_CFC_ (* Continuous Function Chart, elements in execution order *)
(* GYM *)
(* CINEMA *)
(* SHOWER *)
(* SPHERE *)
(* POOL HALL *)
(* TRAINING *)
(* STAIRS *)
#0 fb_sw_01_1_1:FB_ShortLongClick(sw_01_1_1, longPressTimeout)
#1 fb_sw_04_1:FB_ShortLongClick(sw_04_1, longPressTimeout)
#2 fb_sw_07_1_1:FB_ShortLongClick(sw_07_1_1, longPressTimeout)
#3 fb_sw_09_1_1:FB_ShortLongClick(sw_09_1_1, longPressTimeout)
#4 fb_sw_14_1_1:FB_ShortLongClick(sw_14_1_1, longPressTimeout)
#5 fb_sw_01_1_2:FB_ShortLongClick(sw_01_1_2, longPressTimeout)
#6 fb_sw_04_2:FB_ShortLongClick(sw_04_2, longPressTimeout)
#7 fb_sw_07_1_2:FB_ShortLongClick(sw_07_1_2, longPressTimeout)
#8 fb_sw_09_1_2:FB_ShortLongClick(sw_09_1_2, longPressTimeout)
#9 fb_sw_14_1_2:FB_ShortLongClick(sw_14_1_2, longPressTimeout)
#10 fb_sw_05_1:FB_ShortLongClick(sw_05_1, longPressTimeout)
#11 fb_sw_07_2_1:FB_ShortLongClick(sw_07_2_1, longPressTimeout)
#12 fb_sw_09_2_1:FB_ShortLongClick(sw_09_2_1, longPressTimeout)
#13 fb_sw_14_2_1:FB_ShortLongClick(sw_14_2_1, longPressTimeout)
#14 fb_sw_01_2_1:FB_ShortLongClick(sw_01_2_1, longPressTimeout)
#15 fb_sw_05_2:FB_ShortLongClick(sw_05_2, longPressTimeout)
#16 fb_sw_07_2_2:FB_ShortLongClick(sw_07_2_2, longPressTimeout)
#17 fb_sw_09_2_2:FB_ShortLongClick(sw_09_2_2, longPressTimeout)
#18 fb_sw_14_2_2:FB_ShortLongClick(sw_14_2_2, longPressTimeout)
#19 fb_sw_06_1:FB_ShortLongClick(sw_06_1, longPressTimeout)
#20 fb_sw_02_1:FB_ShortLongClick(sw_02_1, longPressTimeout)
#21 fb_sw_09_3_1:FB_ShortLongClick(sw_09_3_1, longPressTimeout)
#22 fb_sw_14_3_1:FB_ShortLongClick(sw_14_3_1, longPressTimeout)
#23 fb_sw_06_2:FB_ShortLongClick(sw_06_2, longPressTimeout)
#24 fb_sw_09_3_2:FB_ShortLongClick(sw_09_3_2, longPressTimeout)
#25 fb_sw_14_3_2:FB_ShortLongClick(sw_14_3_2, longPressTimeout)
#26 fb_sw_02_2:FB_ShortLongClick(sw_02_2, longPressTimeout)
#27 fb_sw_03_1:FB_ShortLongClick(sw_03_1, longPressTimeout)
#28 fb_training01_2_light:FB_Light(-, traning_falling_edge.Q, fb_sw_01_1_1.bLongClick)
#29 OR(fb_sw_01_1_2.bLongClick, fb_sw_05_2.bLongClick, fb_sw_09_3_2.bLongClick)
#30 fb_training_light:FB_Light(-, -, #29)
#31 training02_2_light <= #30
#32 training03_2_light <= #30
#33 OR(#28, #30)
#34 training01_2_light <= #33
#35 traning_falling_edge:F_TRIG(CLK: #30)
#36 OR(traning_falling_edge.Q, traning_reserved_falling_edge.Q)
#37 fb_training01_light:FB_Light(-, #36, fb_sw_01_1_1.bShortClick)
#38 OR(#37, training01_2_light, training02_light)
#39 training01_light <= #38
#40 OR(fb_sw_01_1_2.bShortClick, fb_sw_09_3_2.bShortClick, fb_sw_05_2.bShortClick)
#41 fb_training02_light:FB_Light(-, traning_falling_edge.Q, #40)
#42 traning_reserved_falling_edge:F_TRIG(CLK: #41)
#43 OR(#41, training02_2_light)
#44 training02_light <= #43
#45 fb_training03_light:FB_Light(-, traning_falling_edge.Q, #40)
#46 OR(#45, training03_2_light)
#47 training03_light <= #46
#48 OR(fb_sw_09_2_1.bShortClick, fb_sw_14_2_2.bShortClick)
#49 AND(fb_pool_hall_LED.bLight, fb_pool_hall_spotlight.bLight, pool_hall_all_falling_edge.Q)
#50 fb_pool_hall_LED:FB_Light(pool_hall_all_rising_edge.Q, #49, #48)
#51 pool_hall_ceiling_LED <= #50
#52 pool_hall_LED <= #50
#53 OR(fb_sw_09_2_2.bShortClick, fb_sw_14_2_1.bShortClick)
#54 fb_pool_hall_spotlight:FB_Light(pool_hall_all_rising_edge.Q, #49, #53)
#55 pool_hall_spotlight <= #54
#56 AND(#50, #54)
#57 pool_all_falling_edge:F_TRIG(CLK: #56)
#58 pool_all_rising_edge:R_TRIG(CLK: #56)
#59 OR(fb_sw_09_2_1.bLongClick, fb_sw_14_2_2.bLongClick, fb_sw_09_2_2.bLongClick, fb_sw_14_2_1.bLongClick)
#60 fb_pool_hall_all:FB_Light(pool_all_rising_edge.Q, pool_all_falling_edge.Q, #59)
#61 pool_hall_all_falling_edge:F_TRIG(CLK: #60)
#62 pool_hall_all_rising_edge:R_TRIG(CLK: #60)
#63 OR(fb_sw_09_1_2.bLongClick, fb_sw_14_3_1.bLongClick)
#64 fb_pool_light:FB_Light(-, -, #63)
#65 pool_light <= #102
#66 AND(fb_sw_05_1.bLongClick, fb_sphere_light.bLight, fb_sphere_ceiling_light.bLight)
#67 fb_sphere_light:FB_Light(-, #66, fb_sw_05_1.bLongClick)
#68 sphere_light01 <= #67
#69 sphere_light02 <= #67
#70 fb_sphere_ceiling_light:FB_Light(-, #66, fb_sw_05_1.bShortClick)
#71 OR(#67, #70)
#72 sphere_ceiling_light <= #71
#73 fb_gym_shower01_light:FB_Light(-, -, fb_sw_07_1_2.bShortClick)
#74 gym_shower01_light <= #73
#75 XOR(floor1_tambur3_light, gym_stairs_bra_left)
#76 AND(#75, #101)
#77 OR(fb_sw_02_2.bShortClick, fb_sw_02_2.bLongClick, fb_sw_02_1.bLongClick, #76, fb_sw_01_2_1.bLongClick, fb_sw_01_2_1.bShortClick)
#78 fb_gym_stairs_bra:FB_Light(-, -, #77)
#79 gym_stairs_bra_left <= #78
#80 gym_stairs_bra_right <= #78
#81 fb_gym_shower02_light:FB_Light(-, -, fb_sw_07_1_1.bShortClick)
#82 gym_shower02_light <= #81
#83 fb_gym_stairs_light:FB_Light(-, -, -)
#84 gym_stairs_light <= #83
#85 fb_gym_WC_light:FB_Light(-, -, fb_sw_07_2_1.bShortClick)
#86 gym_WC_light <= #85
#87 fb_gym_corridor_light:FB_Light(-, -, fb_sw_07_2_2.bShortClick)
#88 gym_WC_corridor <= #87
#89 fb_gym01_light:FB_Light(-, gym_falling_edge.Q, fb_sw_14_1_1.bShortClick)
#90 OR(#89, gym02_2_light)
#91 gym01_light <= #90
#92 fb_gym02_light:FB_Light(-, gym_falling_edge.Q, fb_sw_14_1_1.bShortClick)
#93 OR(gym02_2_light, #92)
#94 gym02_light <= #93
#95 fb_gym_cinema_bra:FB_Light(-, -, -)
#96 gym_cinema_bra <= #95
#97 fb_gym_01_2_light:FB_Light(-, -, fb_sw_14_1_1.bLongClick)
#98 gym01_2_light <= #97
#99 gym02_2_light <= #97
#100 gym_falling_edge:F_TRIG(CLK: #97)
#101 OR(sw_floor1_tambur3_short, sw_floor1_tambur3_long)
unconnected input fb_sw_09_2_1.bLongClick
unconnected input fb_sw_14_2_2.bLongClick
#102 OR(sw_09_1_2, sw_14_3_1)
_END_CFC_
END_PROGRAM
ACTION knx_triggers:
	rising_edge_eib_gym01 						(CLK:= eib_gym01);
	rising_edge_eib_gym02 						(CLK:= eib_gym02);
	rising_edge_eib_training01 					(CLK:= eib_training01);
	rising_edge_eib_training02						(CLK:=eib_training02 );
	rising_edge_eib_training03						(CLK:= eib_training03);
	rising_edge_eib_gym_stairs_bra				(CLK:= eib_gym_stairs_bra);
	rising_edge_eib_pool_hall_spotlight				(CLK:=eib_pool_hall_spotlight );
	rising_edge_eib_pool_hall_LED				(CLK:= eib_pool_hall_LED);

	rising_edge_eib_pool_light 					(CLK:= eib_pool_light);
	rising_edge_eib_sphere_ceiling_light 			(CLK:= eib_sphere_ceiling_light);
	rising_edge_eib_sphere_light 					(CLK:= eib_sphere_light);
	rising_edge_eib_gym_cinema_bra 				(CLK:= eib_gym_cinema_bra);
	rising_edge_eib_gym_shower01_light			(CLK:= eib_gym_shower01_light);
	rising_edge_eib_gym_shower02_light			(CLK:= eib_gym_shower02_light);
	rising_edge_eib_gym_corridor_light				(CLK:= eib_gym_corridor_light);
	rising_edge_eib_gym_stairs_light 				(CLK:= eib_gym_stairs_light);

	rising_edge_eib_gym_WC_light 				(CLK:= eib_gym_WC_light);
	rising_edge_eib_training	 					(CLK:= eib_training);
	rising_edge_eib_gym		 					(CLK:= eib_gym);

	falling_edge_eib_gym01 						(CLK:= eib_gym01);
	falling_edge_eib_gym02 						(CLK:= eib_gym02);
	falling_edge_eib_training01 					(CLK:= eib_training01);
	falling_edge_eib_training02						(CLK:=eib_training02 );
	falling_edge_eib_training03						(CLK:= eib_training03);
	falling_edge_eib_gym_stairs_bra				(CLK:= eib_gym_stairs_bra);
	falling_edge_eib_pool_hall_spotlight				(CLK:=eib_pool_hall_spotlight );
	falling_edge_eib_pool_hall_LED				(CLK:= eib_pool_hall_LED);

	falling_edge_eib_pool_light 					(CLK:= eib_pool_light);
	falling_edge_eib_sphere_ceiling_light 			(CLK:= eib_sphere_ceiling_light);
	falling_edge_eib_sphere_light 					(CLK:= eib_sphere_light);
	falling_edge_eib_gym_cinema_bra 				(CLK:= eib_gym_cinema_bra);
	falling_edge_eib_gym_shower01_light			(CLK:= eib_gym_shower01_light);
	falling_edge_eib_gym_shower02_light			(CLK:= eib_gym_shower02_light);
	falling_edge_eib_gym_corridor_light				(CLK:= eib_gym_corridor_light);
	falling_edge_eib_gym_stairs_light 				(CLK:= eib_gym_stairs_light);

	falling_edge_eib_gym_WC_light 				(CLK:= eib_gym_WC_light);
	falling_edge_eib_training	 					(CLK:= eib_training);
	falling_edge_eib_gym		 					(CLK:= eib_gym);
END_ACTION
ACTION outsideLight:
darkOutside_rising_edge(CLK:=bDarkOutside);
IF  bdarkOutside AND (iHour <1 OR iHour>=20) AND iminute=59 THEN
	outside_bigBulbs := TRUE;
	eib_outside_bigBulbs:=TRUE;
	outside_plantsLightning:=TRUE;
	eib_outside_plantsLightning := TRUE;
	outside_smallBulbs := TRUE;
	eib_outside_smallBulbs:= TRUE;
	outside_pingPongTable := FALSE;



ELSE
	outside_bigBulbs := eib_outside_bigBulbs;
	outside_plantsLightning:= eib_outside_plantsLightning;
	outside_smallBulbs := eib_outside_smallBulbs;
	outside_pingPongTable:=eib_outside_pingPongTable;

	IF iHour=2 AND iMinute>=1 AND iMinute<=2 THEN
		outside_bigBulbs := FALSE;
		outside_plantsLightning:=FALSE;
		outside_smallBulbs := FALSE;
		outside_pingPongTable := FALSE;
	END_IF

END_IF;
END_ACTION

(* POU Counters, ST *)
PROGRAM Counters
VAR

	counter_6_KL1408_1_Input : CTU;

	counter_6_KL1408_3_Input	:	CTU;
	counter_6_KL1408_4_Input	:	CTU;
	counter_6_KL1408_5_Input	:	CTU;
	counter_6_KL1408_6_Input	:	CTU;

	counter_6_KL1408_8_Input	:	CTU;
	counter_7_KL1408_1_Input	:	CTU;
	counter_7_KL1408_2_Input	:	CTU;
	counter_7_KL1408_3_Input	:	CTU;
	counter_7_KL1408_4_Input	:	CTU;
	counter_7_KL1408_5_Input	:	CTU;
	counter_7_KL1408_6_Input	:	CTU;
	counter_7_KL1408_7_Input	:	CTU;
	counter_7_KL1408_8_Input	:	CTU;
	counter_8_KL1408_1_Input	:	CTU;
	counter_8_KL1408_2_Input	:	CTU;
	counter_8_KL1408_3_Input	:	CTU;
	counter_8_KL1408_4_Input	:	CTU;
	counter_8_KL1408_5_Input	:	CTU;
	counter_8_KL1408_6_Input	:	CTU;
	counter_8_KL1408_7_Input	:	CTU;
	counter_8_KL1408_8_Input	:	CTU;
	counter_9_KL1408_1_Input	:	CTU;
	counter_9_KL1408_2_Input	:	CTU;
	counter_9_KL1408_3_Input	:	CTU;
	counter_9_KL1408_4_Input	:	CTU;
	counter_9_KL1408_5_Input	:	CTU;
	counter_9_KL1408_6_Input	:	CTU;
	counter_9_KL1408_7_Input	:	CTU;
	counter_9_KL1408_8_Input	:	CTU;
	counter_10_KL1408_1_Input	:	CTU;
	counter_10_KL1408_2_Input	:	CTU;
	counter_10_KL1408_3_Input	:	CTU;
	counter_10_KL1408_4_Input	:	CTU;
	counter_10_KL1408_5_Input	:	CTU;
	counter_10_KL1408_6_Input	:	CTU;
	counter_10_KL1408_7_Input	:	CTU;
	counter_10_KL1408_8_Input	:	CTU;

	sw01 : INT;
	sw02 : INT;
	sw03 : INT;
	sw04 : INT;
	sw05 : INT;
	sw06 : INT;
	sw07 : INT;
	sw08 : INT;
	sw09 : INT;
	sw10 : INT;
	sw11 : INT;
	sw12 : INT;
	sw13 : INT;
	sw14 : INT;
	sw15 : INT;
	sw16 : INT;
	sw17 : INT;
	sw18 : INT;
	sw19 : INT;
	sw20 : INT;
	sw21 : INT;
	sw22 : INT;
	sw23 : INT;
	sw24 : INT;
	sw25 : INT;
	sw26 : INT;
	sw27 : INT;
	sw28 : INT;
	sw29 : INT;
	sw30 : INT;
	sw31 : INT;
	sw32 : INT;
	sw33 : INT;
	sw34 : INT;
	sw35 : INT;
	sw36 : INT;
	sw37 : INT;
	sw38 : INT;
	sw39 : INT;


END_VAR
	counter_6_KL1408_1_Input(CU:= Term_6_KL1408_1_Input, CV=>sw01);

	counter_6_KL1408_3_Input(CU:= Term_6_KL1408_3_Input, CV=>sw02);
	counter_6_KL1408_4_Input(CU:= Term_6_KL1408_4_Input, CV=>sw03);
	counter_6_KL1408_5_Input(CU:= Term_6_KL1408_5_Input, CV=>sw04);





	counter_7_KL1408_3_Input(CU:= Term_7_KL1408_3_Input, CV=>sw09);

	counter_7_KL1408_5_Input(CU:= Term_7_KL1408_5_Input, CV=>sw11);

	counter_7_KL1408_7_Input(CU:= Term_7_KL1408_7_Input, CV=>sw13);












	counter_9_KL1408_2_Input(CU:= Term_9_KL1408_2_Input, CV=>sw24);

	counter_9_KL1408_4_Input(CU:= Term_9_KL1408_4_Input, CV=>sw26);

	counter_9_KL1408_6_Input(CU:= Term_9_KL1408_6_Input, CV=>sw28);

	counter_9_KL1408_8_Input(CU:= Term_9_KL1408_8_Input, CV=>sw30);

	counter_10_KL1408_1_Input(CU:= Term_10_KL1408_1_Input, CV=>sw31);
	counter_10_KL1408_2_Input(CU:= Term_10_KL1408_2_Input, CV=>sw32);
	counter_10_KL1408_3_Input(CU:= Term_10_KL1408_3_Input, CV=>sw33);
	counter_10_KL1408_4_Input(CU:= Term_10_KL1408_4_Input, CV=>sw34);
	counter_10_KL1408_5_Input(CU:= Term_10_KL1408_5_Input, CV=>sw35);
	counter_10_KL1408_6_Input(CU:= Term_10_KL1408_6_Input, CV=>sw36);
	counter_10_KL1408_7_Input(CU:= Term_10_KL1408_7_Input, CV=>sw37);
	counter_10_KL1408_8_Input(CU:= Term_10_KL1408_8_Input, CV=>sw38);
END_PROGRAM
